// Mitsubishi GX Works2 project: water_pump_is_it_ok   PLC: FX3S

// task Task_01 (event TRUE, interval 0, priority 31): POU_01

PROGRAM POU_01
VAR
  fsm_1 : fsm;
  ulazi_1 : ulazi;
  fsm_2 : fsm;
  s_0 : BOOL;
  s_1 : BOOL;
  s_2 : BOOL;
  s_3 : BOOL;
  s_4 : BOOL;
  state : INT;
  goto_1 : BOOL;
  goto_2 : BOOL;
  goto_3 : BOOL;
  goto_4 : BOOL;
  goto_5 : BOOL;
  onnn : BOOL;
  goto_0 : BOOL;
  pokreni : BOOL;
  pumpa : BOOL;
  senzor2 : BOOL;
  senzor1 : BOOL;
  ulazi_2 : ulazi;
  elapsed_time : TIME;
  izlazi_1 : izlazi;
  izlazi_2 : izlazi;
  valve1 : BOOL;
  motor : BOOL;
  puni : BOOL;
  prazni : BOOL;
  valve2 : BOOL;
  ulazi_3 : izlazi;
  izlazi_3 : izlazi;
  alarm : BOOL;
  izlazi_4 : izlazi;
  cnt_done : BOOL;
END_VAR
(* structured ladder/FBD written out as ST: instructions are called as NAME(EN, inputs, outputs); _pN, _eN, _tN stand for wires *)
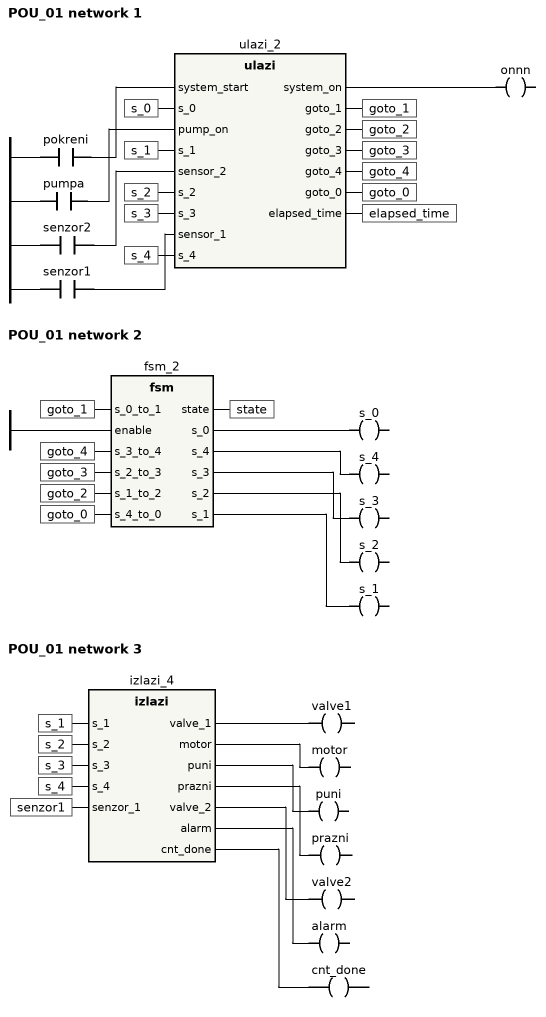
(* network 1 *)
ulazi_2(system_start := pokreni, s_0 := s_0, pump_on := pumpa, s_1 := s_1, sensor_2 := senzor2, s_2 := s_2, s_3 := s_3, sensor_1 := senzor1, s_4 := s_4, goto_1 => goto_1, goto_2 => goto_2, goto_3 => goto_3, goto_4 => goto_4, goto_0 => goto_0, elapsed_time => elapsed_time);
onnn := ulazi_2.system_on;
(* network 2 *)
fsm_2(s_0_to_1 := goto_1, enable := TRUE, s_3_to_4 := goto_4, s_2_to_3 := goto_3, s_1_to_2 := goto_2, s_4_to_0 := goto_0, state => state);
s_0 := fsm_2.s_0;
s_4 := fsm_2.s_4;
s_3 := fsm_2.s_3;
s_2 := fsm_2.s_2;
s_1 := fsm_2.s_1;
(* network 3 *)
izlazi_4(s_1 := s_1, s_2 := s_2, s_3 := s_3, s_4 := s_4, senzor_1 := senzor1);
valve1 := izlazi_4.valve_1;
motor := izlazi_4.motor;
puni := izlazi_4.puni;
prazni := izlazi_4.prazni;
valve2 := izlazi_4.valve_2;
alarm := izlazi_4.alarm;
cnt_done := izlazi_4.cnt_done;
END_PROGRAM

FUNCTION_BLOCK fsm
VAR_OUTPUT
  state : INT;
END_VAR
VAR CONSTANT
  cmp_with_0 : INT;
END_VAR
VAR
  is_eqv : ARRAY [0..2] OF BOOL;
END_VAR
VAR CONSTANT
  cmp_with_1 : INT := 1;
  cmp_with_2 : INT := 2;
  cmp_with_3 : INT := 3;
  cmp_with_4 : INT := 4;
END_VAR
VAR_INPUT
  s_0_to_1 : BOOL;
END_VAR
VAR_OUTPUT
  s_0 : BOOL;
END_VAR
VAR_INPUT
  enable : BOOL;
END_VAR
VAR_OUTPUT
  s_4 : BOOL;
END_VAR
VAR_INPUT
  s_3_to_4 : BOOL;
  s_2_to_3 : BOOL;
END_VAR
VAR_OUTPUT
  s_3 : BOOL;
  s_2 : BOOL;
  s_1 : BOOL;
END_VAR
VAR_INPUT
  s_1_to_2 : BOOL;
  s_4_to_0 : BOOL;
END_VAR
(* structured ladder/FBD written out as ST: instructions are called as NAME(EN, inputs, outputs); _pN, _eN, _tN stand for wires *)
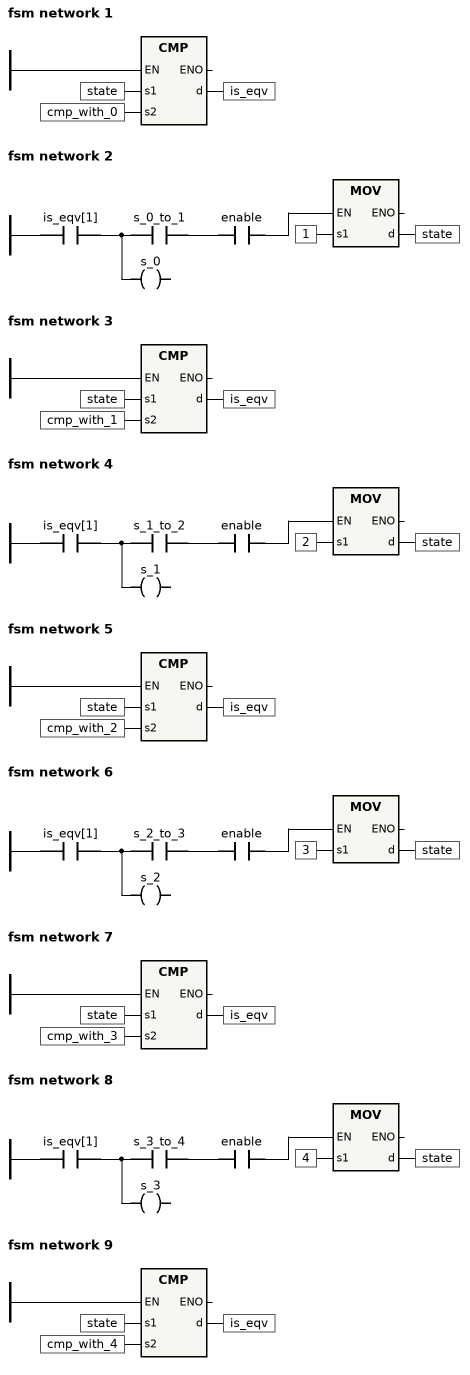
(* network 1 *)
CMP(TRUE, state, cmp_with_0, is_eqv);
(* network 2 *)
MOV(is_eqv[1] AND s_0_to_1 AND enable, 1, state);
s_0 := is_eqv[1];
(* network 3 *)
CMP(TRUE, state, cmp_with_1, is_eqv);
(* network 4 *)
MOV(is_eqv[1] AND s_1_to_2 AND enable, 2, state);
s_1 := is_eqv[1];
(* network 5 *)
CMP(TRUE, state, cmp_with_2, is_eqv);
(* network 6 *)
MOV(is_eqv[1] AND s_2_to_3 AND enable, 3, state);
s_2 := is_eqv[1];
(* network 7 *)
CMP(TRUE, state, cmp_with_3, is_eqv);
(* network 8 *)
MOV(is_eqv[1] AND s_3_to_4 AND enable, 4, state);
s_3 := is_eqv[1];
(* network 9 *)
CMP(TRUE, state, cmp_with_4, is_eqv);
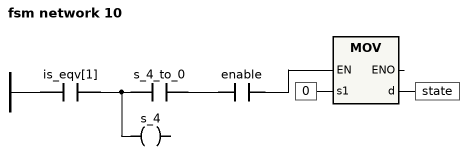
(* network 10 *)
MOV(is_eqv[1] AND s_4_to_0 AND enable, 0, state);
s_4 := is_eqv[1];
END_FUNCTION_BLOCK

FUNCTION_BLOCK ulazi
VAR_INPUT
  system_start : BOOL;
END_VAR
VAR_OUTPUT
  system_on : BOOL;
END_VAR
VAR
  system_off : BOOL;
END_VAR
VAR_INPUT
  s_0 : BOOL;
  pump_on : BOOL;
END_VAR
VAR_OUTPUT
  goto_1 : BOOL;
END_VAR
VAR_INPUT
  s_1 : BOOL;
  sensor_2 : BOOL;
END_VAR
VAR_OUTPUT
  goto_2 : BOOL;
END_VAR
VAR_INPUT
  s_2 : BOOL;
END_VAR
VAR
  TON_1 : TON;
END_VAR
VAR CONSTANT
  pause : TIME := T#10s;
END_VAR
VAR_OUTPUT
  goto_3 : BOOL;
END_VAR
VAR_INPUT
  s_3 : BOOL;
  sensor_1 : BOOL;
END_VAR
VAR_OUTPUT
  goto_4 : BOOL;
END_VAR
VAR_INPUT
  s_4 : BOOL;
END_VAR
VAR_OUTPUT
  goto_0 : BOOL;
  elapsed_time : TIME;
END_VAR
(* structured ladder/FBD written out as ST: instructions are called as NAME(EN, inputs, outputs); _pN, _eN, _tN stand for wires *)
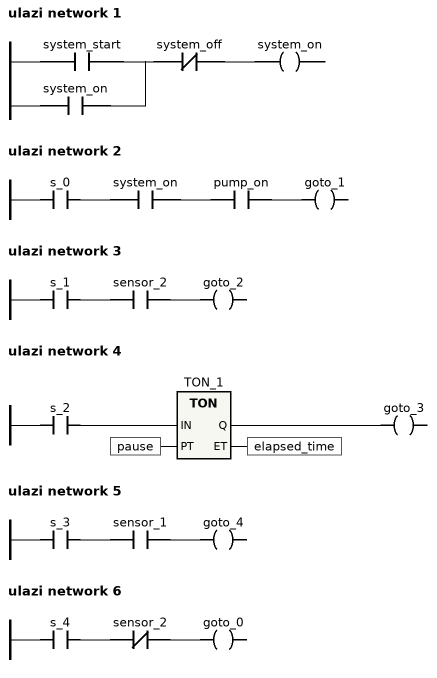
(* network 1 *)
system_on := (system_start OR system_on) AND NOT system_off;
(* network 2 *)
goto_1 := s_0 AND system_on AND pump_on;
(* network 3 *)
goto_2 := s_1 AND sensor_2;
(* network 4 *)
TON_1(IN := s_2, PT := pause, ET => elapsed_time);
goto_3 := TON_1.Q;
(* network 5 *)
goto_4 := s_3 AND sensor_1;
(* network 6 *)
goto_0 := s_4 AND NOT sensor_2;
END_FUNCTION_BLOCK

FUNCTION_BLOCK izlazi
VAR_INPUT
  s_1 : BOOL;
  s_2 : BOOL;
  s_3 : BOOL;
END_VAR
VAR_OUTPUT
  valve_1 : BOOL;
  motor : BOOL;
END_VAR
VAR_INPUT
  s_4 : BOOL;
END_VAR
VAR_OUTPUT
  puni : BOOL;
  prazni : BOOL;
  valve_2 : BOOL;
END_VAR
VAR_INPUT
  senzor_1 : BOOL;
END_VAR
VAR_OUTPUT
  alarm : BOOL;
END_VAR
VAR
  cnt_cycles_1 : cnt_cycles;
END_VAR
VAR_OUTPUT
  cnt_done : BOOL;
END_VAR
(* structured ladder/FBD written out as ST: instructions are called as NAME(EN, inputs, outputs); _pN, _eN, _tN stand for wires *)
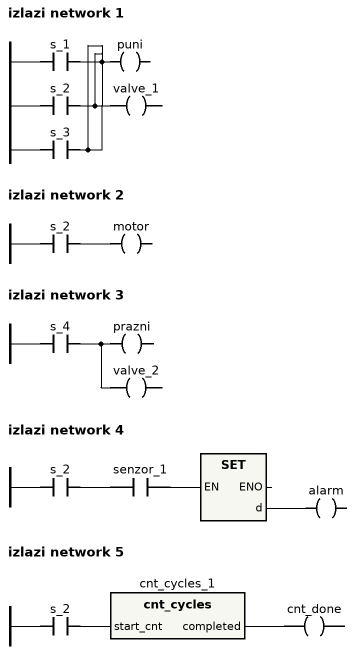
(* network 1 *)
_p1 := s_1 OR s_2 OR s_3;
puni := _p1;
valve_1 := _p1;
(* network 2 *)
motor := s_2;
(* network 3 *)
prazni := s_4;
valve_2 := s_4;
(* network 4 *)
SET(s_2 AND senzor_1, _t1);
alarm := _t1;
(* network 5 *)
cnt_cycles_1(start_cnt := s_2);
cnt_done := cnt_cycles_1.completed;
END_FUNCTION_BLOCK

FUNCTION_BLOCK cnt_cycles
VAR_INPUT
  start_cnt : BOOL;
END_VAR
VAR
  state : INT;
END_VAR
VAR CONSTANT
  add_1 : INT := 1;
  cmp_with_5 : INT := 5;
END_VAR
VAR
  is_done : ARRAY [0..2] OF BOOL;
END_VAR
VAR_OUTPUT
  completed : BOOL;
END_VAR
VAR
  is_eqv : ARRAY [0..2] OF BOOL;
END_VAR
(* structured ladder/FBD written out as ST: instructions are called as NAME(EN, inputs, outputs); _pN, _eN, _tN stand for wires *)
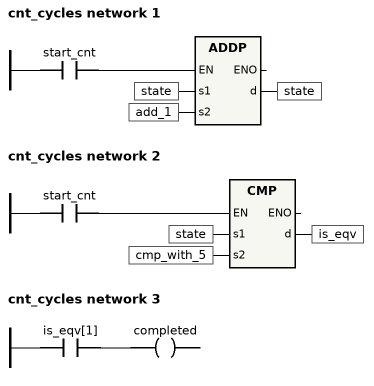
(* network 1 *)
ADDP(start_cnt, state, add_1, state);
(* network 2 *)
CMP(start_cnt, state, cmp_with_5, is_eqv);
(* network 3 *)
completed := is_eqv[1];
END_FUNCTION_BLOCK
